// LS Electric XG5000 project: pppp
// PLC NewPLC

PROGRAM NewProgram (task: Scan Program)

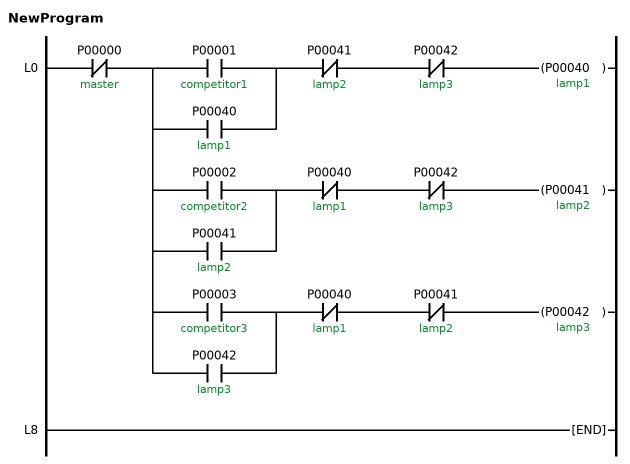
; L0
LOAD NOT  P00000	// master
MPUSH
LOAD      P00001	// competitor1
OR        P00040	// lamp1
AND LOAD
AND NOT   P00041	// lamp2
AND NOT   P00042	// lamp3
OUT       P00040	// lamp1
MLOAD
LOAD      P00002	// competitor2
OR        P00041	// lamp2
AND LOAD
AND NOT   P00040	// lamp1
AND NOT   P00042	// lamp3
OUT       P00041	// lamp2
MPOP
LOAD      P00003	// competitor3
OR        P00042	// lamp3
AND LOAD
AND NOT   P00040	// lamp1
AND NOT   P00041	// lamp2
OUT       P00042	// lamp3
; L8
END